FUNCTION_BLOCK PUBLIC FB_CDPlayer
VAR_OUTPUT
	bPlayerActive		: BOOL;
	byVolume			: BYTE;
	byTrack				: UINT;
END_VAR

PROPERTY PUBLIC PlayerActive : BOOL
GET
PlayerActive := bPlayerActive;
END_GET
END_PROPERTY

METHOD PUBLIC SetTrack : BOOL
VAR_INPUT
	byNewTrack			: UINT;
END_VAR
byTrack := byNewTrack;
END_METHOD

METHOD PUBLIC SetVolume : BOOL
VAR_INPUT
	byNewVolume 		: BYTE;
END_VAR
byVolume := byNewVolume;
END_METHOD

METHOD PUBLIC Start
bPlayerActive := true;
END_METHOD

METHOD PUBLIC Stop
bPlayerActive := FALSE;
END_METHOD

PROPERTY PUBLIC Track : UINT
GET
Track := byTrack;
END_GET
END_PROPERTY

PROPERTY PUBLIC Volume : BYTE
GET
Volume := byVolume;
END_GET
END_PROPERTY

END_FUNCTION_BLOCK

(* stored: Version 1.1.0.1, ProductVersion 3.1.4020.3
   POU FB_CDPlayer: Id {e5938590-1890-43a0-ba86-32547ab377e2}, SpecialFunc None
   Property PlayerActive: Id {5747ae8d-4a33-4113-9fd7-8425111c955f}
   Get Get: Id {22b85649-b7cf-4b58-b014-46b33f3f2cea}
   Method SetTrack: Id {4e5634f0-9545-430f-86b8-452bc4855175}
   Method SetVolume: Id {eccc8046-24a1-4940-82a7-bde5c3e6c0ab}
   Method Start: Id {bdc89d87-e6d0-409f-9392-70820315cfad}
   Method Stop: Id {e998b74b-1a66-4831-b792-c8f260a073f3}
   Property Track: Id {b0a7ebff-501f-4cac-8dfd-fc0417cc4c86}
   Get Get: Id {ab8c61dd-0b4c-42b1-9ad5-ddc83fc36787}
   Property Volume: Id {ce5fac73-4811-427f-aabd-cccf1f8f19c1}
   Get Get: Id {4e7aa514-d712-4467-8f60-745f5909e0e6} *)
